FUNCTION_BLOCK EventLogger
VAR
	EventBuffer : ARRAY[1..Maxinum_size_event_buffer] OF ST_Event;
	CurrentEventBufferIndex : INT := 0;
	
	_PersistentEventStorage : I_PersistentEventStorage;
END_VAR
VAR CONSTANT
	Maxinum_size_event_buffer : INT := 100;
END_VAR

(* Returns TRUE if add was succesful and FALSE if buffer is full *)
METHOD PUBLIC AddEvent : BOOL
VAR_INPUT
	eEventType : E_EventType;
	eEventSeverity : TcEventSeverity;
	nEventIdentity : UDINT;
	sEventText : STRING(255);
END_VAR
IF NOT IsEventBufferFull() THEN
	CurrentEventBufferIndex := CurrentEventBufferIndex + 1;
	EventBuffer[CurrentEventBufferIndex].eEventType := eEventType;
	EventBuffer[CurrentEventBufferIndex].eEventSeverity := eEventSeverity;
	EventBuffer[CurrentEventBufferIndex].nEventIdentity := nEventIdentity;
	EventBuffer[CurrentEventBufferIndex].sEventText := sEventText;
	F_UpdateEventTimestampWithSystemTime(stEvent := EventBuffer[CurrentEventBufferIndex]);
	AddEvent := TRUE;
ELSE
	AddEvent := FALSE;		
END_IF


// Event Persistently

_PersistentEventStorage.StoreEvent(stEvent := EventBuffer[CurrentEventBufferIndex]);
END_METHOD

METHOD FB_init : BOOL
VAR_INPUT
	bInitRetains : BOOL; // if TRUE, the retain variables are initialized (warm start / cold start)
	bInCopyCode : BOOL;  // if TRUE, the instance afterwards gets moved into the copy code (online change)
	
	iPersistentEventStorage : I_PersistentEventStorage;
END_VAR
_PersistentEventStorage := iPersistentEventStorage;
END_METHOD

METHOD PRIVATE IsEventBufferFull : BOOL
IF (CurrentEventBufferIndex + 1) > Maxinum_size_event_buffer THEN 
	IsEventBufferFull := TRUE;
ELSE 
	IsEventBufferFull := FALSE;
END_IF
END_METHOD

END_FUNCTION_BLOCK

(* stored: Version 1.1.0.1, ProductVersion 3.1.4024.12
   POU EventLogger: Id {ec4c6b28-9f52-423e-8848-9943ea774b7a}, SpecialFunc None
   Method AddEvent: Id {3eebf9f1-d8c3-4a31-8cf3-9767513c6e54}
   Method FB_init: Id {37f92d89-e580-4252-8dd3-8fb51d240786}
   Method IsEventBufferFull: Id {9c7b50ce-08d3-4e03-965d-9fdb6985eed0} *)
